// TwinCAT 3 PLC project Proj_Ueb_sw01_Rs232
// ProgramVersion: 3.1.4023.0
// libraries:
//   Tc2_Standard, * (Beckhoff Automation GmbH)
//   Tc2_System, * (Beckhoff Automation GmbH)
//   Tc3_Module, * (Beckhoff Automation GmbH)
// project tree:
//   DUTs/ St_RS232Word.TcDUT
//   / PlcTask.TcTTO
//   POUs/ FUN_ParseStatusWord.TcPOU, MAIN.TcPOU
// (motion and I/O tree: see PLC project proj_sw01)
// real-time tasks:
//   TASK PlcTask: cycle T#10ms, priority 20, ADS port 350
//   TASK PlcTask1: cycle T#10ms, priority 21, ADS port 351
//   TASK PlcTask2: cycle T#10ms, priority 22, ADS port 352
// variable links:

CONFIGURATION Proj_Ueb_sw01_Rs232
    RESOURCE PLC ON TwinCAT3
        TASK PlcTask(INTERVAL := T#10ms, PRIORITY := 22);
        PROGRAM MAIN WITH PlcTask : MAIN;
    END_RESOURCE
END_CONFIGURATION

// ---- DUTs/St_RS232Word.TcDUT
TYPE St_RS232Word :
STRUCT
	inLength			: INT;
	overrunError		: BOOL;
	framingError		: BOOL;
	parityError 		: BOOL;
	bufferFull			: BOOL;
	initAccepted		: BOOL;
	recieveAccepted		: BOOL;
	transmitAccepted	: BOOL;
END_STRUCT
END_TYPE

// ---- POUs/MAIN.TcPOU
PROGRAM MAIN
VAR
	myWord			: WORD := 16#5D7A;
	myResult		: WORD;
	myDword			: DWORD;
	parsedWord		: St_RS232Word;
END_VAR

myResult := SHR(myWord, 3);
myDword  := SHL(myWord, 3);

myDword  := myDword OR 16#F0000000;


parsedWord := FUN_ParseStatusWord(16#1D06);
parsedWord := FUN_ParseStatusWord(16#534C);
parsedWord := FUN_ParseStatusWord(16#C705);

END_PROGRAM

// ---- POUs/FUN_ParseStatusWord.TcPOU
FUNCTION FUN_ParseStatusWord : St_RS232Word
VAR_INPUT
	w_Status			: WORD;
END_VAR
VAR
	parsedWord			: St_RS232Word;
END_VAR

// extract data : shift to right and convert to Integer
parsedWord.inLength := WORD_TO_INT( SHR(w_Status, 8) );

// extract flag bits
parsedWord.overrunError 		:= (w_Status AND 2#100_0000) > 0;	
parsedWord.framingError 		:= (w_Status AND 2#010_0000) > 0;	
parsedWord.parityError 		:= (w_Status AND 2#001_0000) > 0;	
parsedWord.bufferFull 			:= (w_Status AND 2#000_1000) > 0;	
parsedWord.initAccepted		:= (w_Status AND 2#000_0100) > 0;	
parsedWord.recieveAccepted 	:= (w_Status AND 2#000_0010) > 0;	
parsedWord.transmitAccepted	:= (w_Status AND 2#000_0001) > 0;	

FUN_ParseStatusWord := parsedWord;

END_FUNCTION
